FUNCTION_BLOCK Station001 EXTENDS TcoCore.TcoObject 
VAR
	_components : Station001_Components(THIS^);
	
	_groundMode : Station001_GroundMode(THIS^, eRestoreMode.None);
	_automatMode : Station001_AutomatMode(THIS^, eRestoreMode.None);
	_swiftSequence   : Station001_Swift(THIS^, eRestoreMode.None);
	
	_groundModeTask : TcoCore.TcoTask(THIS^);
	_automatModeTask : TcoCore.TcoTask(THIS^);
	_serviceModeTask : TcoCore.TcoTask(THIS^);
	_swiftModeTask : TcoCore.TcoTask(THIS^);
	
	
	_processRecipies : ProcessDataManager(THIS^); 
    _processTraceabilty : ProcessDataManager(THIS^);
	_technologicalDataManager : TechnologicalDataManager(THIS^);
	_currentMode : enumModes := enumModes.Idle;
	_checkers : Checkers(THIS^);
	
	_externalToken : STRING;
	_externalTokenPresence : BOOL;
END_VAR

_components();
_processRecipies();
_processTraceabilty();
_technologicalDataManager();

ServiceMode();
GroundMode();
AutomatMode();


IF(_swiftModeTask.Execute()) THEN
	Messenger.Trace('Service mode active');	
	_automatModeTask.Restore();
	_groundModeTask.Restore();
	_groundMode.Restore();
	_automatMode.Restore();
	_serviceModeTask.Restore();
	_swiftSequence.Run();
	_currentMode := enumModes.Idle;
END_IF

METHOD AutomatMode : BOOL
VAR_INPUT
END_VAR
_automatModeTask.Enabled := _groundModeTask.Done;

IF(_automatModeTask.Execute()) THEN
	Messenger.Trace('Automat mode active');
	_serviceModeTask.Abort();
	_automatMode.Run();
	_currentMode := enumModes.Automat;
END_IF
END_METHOD

PROPERTY Checkers : REFERENCE TO Checkers
GET
Checkers REF= _checkers;
END_GET
END_PROPERTY

PROPERTY Components : REFERENCE TO Station001_Components
GET
Components REF= _components;
END_GET
END_PROPERTY

METHOD GroundMode : BOOL
VAR_INPUT
END_VAR
IF(_groundModeTask.Execute()) THEN
	Messenger.Trace('Ground position mode active');
	_serviceModeTask.Restore();
	_automatModeTask.Restore();
	_automatMode.Restore();
	_groundMode.Run();
	_groundModeTask.DoneWhen(_groundMode.CurrentStep.ID = 300);
	IF _groundModeTask.Done THEN
		_groundMode.Restore();
	END_IF
	_currentMode := enumModes.Ground;
END_IF
END_METHOD

PROPERTY ProcessRecepie : REFERENCE TO ProcessDataManager
GET
ProcessRecepie REF= _processRecipies;
END_GET
END_PROPERTY

PROPERTY ProcessTraceabilty : REFERENCE TO ProcessDataManager
GET
ProcessTraceabilty REF= _processTraceabilty;
END_GET
END_PROPERTY

PROPERTY  ProductionData : REFERENCE TO Station001_ProductionData
GET
ProductionData REF= _processTraceabilty._data;
END_GET
END_PROPERTY

METHOD ServiceMode
VAR_INPUT
END_VAR
IF(_serviceModeTask.Execute()) THEN
	Messenger.Trace('Service mode active');	
	_automatModeTask.Restore();
	_groundModeTask.Restore();
	_groundMode.Restore();
	_automatMode.Restore();
	_components.Service();
	_currentMode := enumModes.Service;
END_IF
END_METHOD

PROPERTY TechnologicalDataManager : REFERENCE TO TechnologicalDataManager
GET
TechnologicalDataManager REF= _technologicalDataManager;
END_GET
END_PROPERTY

END_FUNCTION_BLOCK

(* stored: Version 1.1.0.1, ProductVersion 3.1.4024.9
   POU Station001: Id {3d3ca50a-cd66-4945-a21d-285298b2ba20}, SpecialFunc None
   Method AutomatMode: Id {06ac0ea5-9bba-426c-9f50-97641acc5f1f}
   Property Checkers: Id {9cd1367e-8bb5-450c-807d-957b9f194b6b}
   Get Get: Id {92f1b29e-36ad-4210-8aba-8d49ce2d0eba}
   Property Components: Id {9262f3ea-0398-44d7-8cae-cfc2e667ba08}
   Get Get: Id {dacd1503-9951-4498-890f-66fd2c5babde}
   Method GroundMode: Id {d9df9b20-93b2-469b-9293-a125a7afb90b}
   Property ProcessRecepie: Id {b1b59222-8dec-42af-9785-f7a41fdb1f30}
   Get Get: Id {7693ce53-8625-4a27-a0d9-a13a48b1061c}
   Property ProcessTraceabilty: Id {53bc7e1b-e1d9-4700-b7ae-13b971dd1d3f}
   Get Get: Id {f0b6082c-910f-4dff-a364-02438a23363f}
   Property ProductionData: Id {fe3a70b9-7cb2-4332-97ec-d5340b743354}
   Get Get: Id {bea63141-a4c5-4e30-9707-f7de4dfe42cd}
   Method ServiceMode: Id {249d59c0-627f-4b64-aec6-5c46efb6257a}
   Property TechnologicalDataManager: Id {4fd8d00a-71e1-4167-bc5c-91bc32c791d7}
   Get Get: Id {2a909450-f811-4a6b-9ceb-c37e0584a44f} *)
